(* IEC 61131-3 sources: HappyLearnCodesys/content/softmotion/CNC07_Subprogram, 3 files *)

(* ---- GVL.st ---- *)
VAR_GLOBAL
	g_x: REAL:=400;
	g_y: REAL:=200;
END_VAR

VAR_GLOBAL CONSTANT
	gc_dwCycle : DWORD := 4000;
END_VAR

(* ---- CNC.st ---- *)
PROGRAM CNC
VAR
	iState: INT;
	pX, pY, pZ: MC_Power;

	ipo: SMC_Interpolator;
	trafo: SMC_TRAFO_Gantry3;
	trafof: SMC_TRAFOF_Gantry3D;
	cabpX, 	cabpY, 	cabpZ: SMC_ControlAxisByPos;

END_VAR

pX(
	Enable:=TRUE ,
	bRegulatorOn:=TRUE ,
	bDriveStart:=TRUE ,
	Axis:=AxisX);
pY(
	Enable:=TRUE ,
	bRegulatorOn:=TRUE ,
	bDriveStart:=TRUE ,
	Axis:=AxisY);
pZ(
	Enable:=TRUE ,
	bRegulatorOn:=TRUE ,
	bDriveStart:=TRUE ,
	Axis:=AxisZ);

CASE iState OF
0:
	IF pX.Status AND pY.Status AND pZ.Status THEN
		iState:=100;
	END_IF
100:
	Interpolation();
END_CASE

(* ---- CNC_PreparePath.st ---- *)
PROGRAM CNC_PreparePath
VAR_INPUT
	xStart: BOOL;
	sFileName: STRING := 'Application/CNC2Main.cnc';
END_VAR
VAR_OUTPUT
	xStartIpo: BOOL;
	poqPath: Pointer to SMC_Outqueue;
END_VAR
VAR
	iState: INT;
	rncf2 : SMC_ReadNCFile2 := (aSubProgramDirs := ['Application/']);
	nci : SMC_NCInterpreter;
	cv : SMC_CheckVelocities;
	aBufInterpreter : ARRAY[0..99] OF SMC_GeoInfo ;
    dnccs : SMC_DisplayNCCallstack;

	sentenc: SMC_GSentenceQueue;
	asv : ARRAY[0..1] OF SMC_SingleVar := [
  	(strVarName := 'G_X', eVarType := SMC_TYPE_REAL, pAdr := ADR(g_x)),
  	(strVarName := 'G_Y', eVarType := SMC_TYPE_REAL, pAdr := ADR(g_y))];
	vl : SMC_VarList := (wNumberVars := 2, psvVarList := ADR(asv[0]));
END_VAR

poqPath := cv.poqDataOut;
dnccs(
    csi := nci.CallstackInfo,
    ipo := CNC.ipo,
    Enable := TRUE);

CASE iState OF
0:	// idle
	IF xStart THEN
		iState:=10;
		xStartIpo := FALSE;
		rncf2(bExecute:=FALSE);
		nci(bExecute:=FALSE,sentences := rncf2.sentences);
		cv(bExecute:=FALSE);
		xStart:=FALSE;
	END_IF

10:	// start reading and processing
	rncf2(
        bExecute:=TRUE ,
		sFileName:=sFileName ,
		pvl:= ADR(vl));

	nci(
        bExecute:=TRUE ,
		sentences := rncf2.sentences,
		nSizeOutQueue:=SIZEOF(aBufInterpreter) ,
		pbyBufferOutQueue:=ADR(aBufInterpreter),
        bEnableSyntaxChecks:= TRUE,
        eOriConv:= SMC_ORI_CONVENTION.ZYZ);

	cv(
        bExecute:= TRUE,
		poqDataIn:=nci.poqDataOut);

	xStartIpo := TRUE;
	IF NOT cv.bBusy THEN
		iState:=0;
	END_IF
END_CASE
